FUNCTION_BLOCK AlarmViewLogger IMPLEMENTS EventLogger
VAR_INPUT
END_VAR
VAR_OUTPUT
END_VAR
VAR
  events: ARRAY[1..Properties.ALARM_VIEW_NUM_EVENTS] OF EventMessageHMI;
  empty_message: EventMessageHMI;
  _level: EventLevel;
  act_time: TIMESTRUCT;
  act_time_str: STRING(255);
  format_string: FB_FormatString;
  _datetime_format: STRING(255) := '%4.0f-%02.0f-%02.0f %02.0f:%02.0f:%02.0f.%03.0f';
END_VAR

METHOD clear_event_message
VAR_INPUT
	id: INT;
END_VAR
VAR
  index: INT;
  filldata: EventMessageHMI;
END_VAR
IF event_in_table(id:=id) THEN
  index := event_index(id:=id);
  
  remove_field_from_array(
    index_to_remove:=index,
    size_filldata:=SIZEOF(filldata),
    adr_filldata:=ADR(filldata),
    size_memory_buffer:=SIZEOF(events),
    adr_memory_buffer:=ADR(events));
END_IF
END_METHOD

PROPERTY PUBLIC datetime_format : STRING(255)
GET
datetime_format := _datetime_format;
END_GET
SET
_datetime_format := datetime_format;
END_SET
END_PROPERTY

METHOD PRIVATE event_in_table : BOOL
VAR_INPUT
  id: INT;
END_VAR
event_in_table := event_index(id) > 0;
END_METHOD

METHOD PRIVATE event_index : INT
VAR_INPUT
  id: INT;
END_VAR
VAR
  i: INT;
END_VAR
FOR i:=1 TO Properties.ALARM_VIEW_NUM_EVENTS DO
  // there are no gaps between events, so it is safe to assume
  // that the first empty event is the end
  IF events[i].id = 0 THEN
    EXIT;
	END_IF
  
  IF events[i].id := id THEN
    event_index := i;
    EXIT;
	END_IF
END_FOR
END_METHOD

PROPERTY PUBLIC level : EventLevel
GET
level := _level;
END_GET
SET
_level := level;
END_SET
END_PROPERTY

METHOD PUBLIC reset
VAR_INPUT
  execute: BOOL;
END_VAR
VAR
  i: INT;
END_VAR
VAR_INST
  r_execute: R_TRIG;
END_VAR
r_execute(CLK:=execute);
IF r_execute.Q THEN
  logging.reset_events_and_messages();
  FOR i:=1 TO Properties.ALARM_VIEW_NUM_EVENTS DO
    events[i] := empty_message;
	END_FOR
END_IF
END_METHOD

METHOD run
VAR_INPUT
	act_time	: Tc2_Utilities.TIMESTRUCT;
END_VAR
VAR_INST
  year: REAL;
  month: REAL;
  day: REAL;
  hour: REAL;
  minute: REAL;
  second: REAL;
  millisecond: REAL;
END_VAR
VAR
END_VAR
THIS^.act_time := act_time;
// ugly hack. have to convert numbers to real because the format specification
// only allows leading zeros on types f, e and s
year := TO_REAL(act_time.wYear);
month := TO_REAL(act_time.wMonth);
day := TO_REAL(act_time.wDay);
hour := TO_REAL(act_time.wHour);
minute := TO_REAL(act_time.wMinute);
second := TO_REAL(act_time.wSecond);
millisecond := TO_REAL(act_time.wMilliseconds);
format_string(
  sFormat:=datetime_format,
  arg1:=F_REAL(year),
  arg2:=F_REAL(month),
  arg3:=F_REAL(day),
  arg4:=F_REAL(hour),
  arg5:=F_REAL(minute),
  arg6:=F_REAL(second),
  arg7:=F_REAL(millisecond),
  sOut=>act_time_str);
END_METHOD

METHOD submit_event_message
VAR_IN_OUT
	ev: EventMessage;
END_VAR
VAR_INST
  ev_hmi: EventMessageHMI;
END_VAR
IF ev.level >= level THEN
  ev_hmi.id := ev.id;
  ev_hmi.level := ev.level;
  ev_hmi.message := ev.message.str;
  ev_hmi.path := ev.path.str;
  ev_hmi.timestamp := act_time_str;
  put_new_data_at_start(SIZEOF(ev_hmi), ADR(ev_hmi), SIZEOF(events), ADR(events));
END_IF
END_METHOD

END_FUNCTION_BLOCK

(* stored: Version 1.1.0.1, ProductVersion 3.1.4022.18
   POU AlarmViewLogger: Id {b90ec479-5310-4abf-adeb-bad2f6cff5d7}, SpecialFunc None
   Method clear_event_message: Id {aeb1148d-756f-4577-a075-dfc54b0c3260}
   Property datetime_format: Id {86e3183d-d03c-4a29-977d-60d740970beb}
   Get Get: Id {90f39645-2cc5-49a9-8665-cc0db8146f32}
   Set Set: Id {157f0eef-4b71-4290-a80c-a58eddb99984}
   Method event_in_table: Id {284b3227-559e-49bb-9754-2f0306e475b3}
   Method event_index: Id {d4a08f6d-cd9c-47e6-9893-a9926832b62a}
   Property level: Id {d383f47b-c7e8-4ec6-a222-5dd0cc857a16}
   Get Get: Id {9cdae7c4-013f-4597-aa67-3b4fbf2062b3}
   Set Set: Id {b5c89708-4977-48f9-81fe-b00e169d114a}
   Method reset: Id {b05a7595-f32b-4d18-b444-ab46d22f0168}
   Method run: Id {94d44a78-563d-472f-bc28-9cbe9d075abe}
   Method submit_event_message: Id {7614287c-c461-4ecf-835d-82cb246574a4} *)
